{attribute 'qualified_only'}
VAR_GLOBAL
END_VAR

(* stored: Version 1.1.0.1, ProductVersion 3.1.4024.12
   GVL G_Enables: Id {a1c2cbb9-0c9a-4461-9d39-fa0eb030f6b4} *)
